# EPICS alarm handler configuration: apps/alhConfig/svtVoltage.alhConfig
#===============================================================================
# SVT Voltage Alarm Config
#===============================================================================

GROUP NULL VOLTAGE
$GUIDANCE
See SVT Ops manual sections relating to voltages.
$END

INCLUDE VOLTAGE /usr/clas12/hps/prod/apps/alhConfig/svtBias.alhConfig
INCLUDE VOLTAGE /usr/clas12/hps/prod/apps/alhConfig/svtLV.alhConfig
INCLUDE VOLTAGE /usr/clas12/hps/prod/apps/alhConfig/svtFlangeLV.alhConfig
